FUNCTION_BLOCK SecondOrderLag
VAR_INPUT
	d : 	REAL;
	w : 	REAL;
	h : 	REAL;
	x : 	REAL;
END_VAR
VAR_OUTPUT
	y : 	REAL;
END_VAR
VAR
	xm : 	REAL;
	xmm : 	REAL;
	ym :	REAL;
	ymm : 	REAL;
END_VAR

y := xmm*w*w*h*h-ym*(-2+2*d*w*h)-ymm*(1-2*d*w*h+w*w*h*h);
ymm := ym;
ym := y;
xmm := xm;
xm := x;

END_FUNCTION_BLOCK

(* stored: Version 1.1.0.1, ProductVersion 3.1.4024.13
   POU SecondOrderLag: Id {fae0f55b-d1a1-4298-a16e-43964164497a}, SpecialFunc None *)
